(* Logix 5000 project; controller MECHATRONICS_FINAL 1769-L16ER-BB1B rev 32.11; software revision 32.00 *)

TASK MainTask (continuous, watchdog 500 ms) : MainProgram

MODULES
   Local : 1769-L16ER-BB1B (PointIO 0, rev 32.11)
      Discrete_IO : Embedded (PointIO 1, rev 32.11, Output RPI 20 ms)
END_MODULES

PROGRAM MainProgram   (* main routine MainRoutine *)
VAR
   Brakes : BOOL;
   CurrentFloor : DINT := 1;
   DoorOpen : BOOL;
   ElevatorButton : BOOL;
   EntireGarageFull : BOOL;
   FloorCapacity : INT[6] := ([0] := 8, [1] := 8, [2] := 8, [3] := 8, [4] := 8, [5] := 8);
   index : DINT;
   MotorDown : BOOL;
   MotorDownOS : BOOL;
   MotorDownTimer : TIMER := (PRE := 5000);
   MotorUp : BOOL;
   MotorUpOS : BOOL;
   MotorUpTimer : TIMER := (PRE := 5000);
   RequestArray : INT[5];
   RequestButton1 : BOOL;
   RequestButton2 : BOOL;
   RequestButton3 : BOOL;
   RequestButton4 : BOOL;
   RequestButtonBase : BOOL;
   RequestInProgress : BOOL;
   RequestOut1 : BOOL;
   RequestOut2 : BOOL;
   RequestOut3 : BOOL;
   RequestOut4 : BOOL;
   SequenceStep : DINT;
   TempVal : DINT;
   VehicleInPlace : BOOL;
   WaitTimer : TIMER := (PRE := 30000);
END_VAR

ROUTINE MainRoutine   (* ladder *)
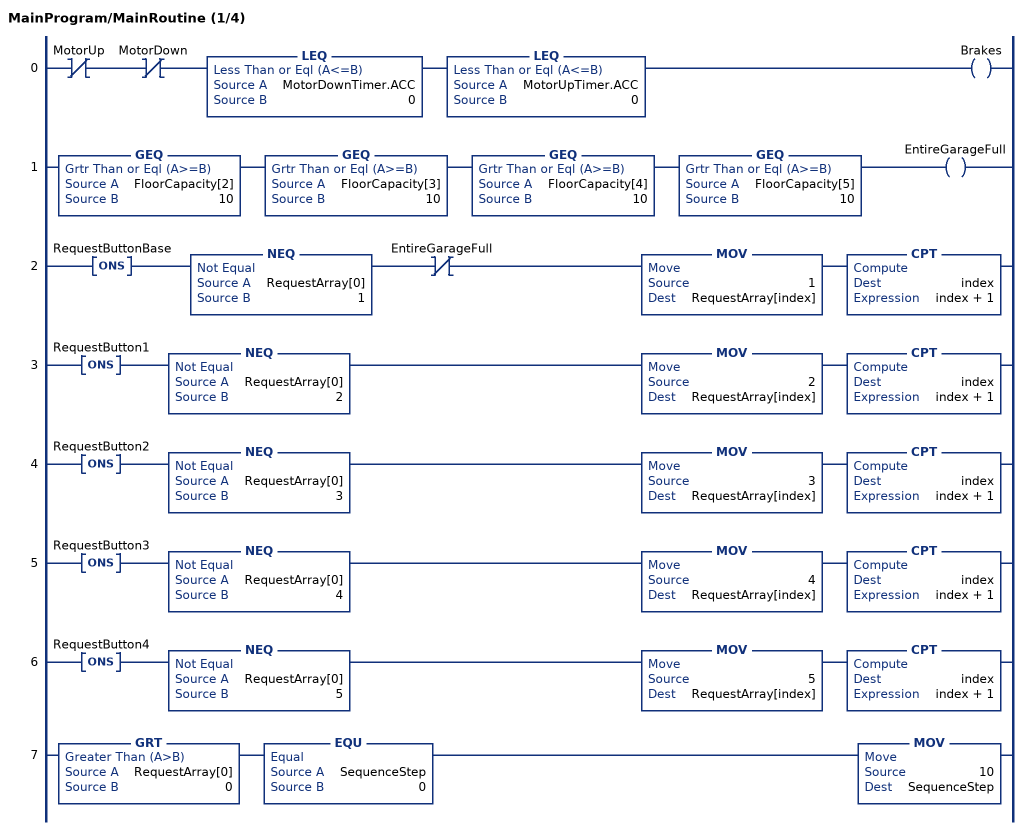
   0: XIO(MotorUp)XIO(MotorDown)LEQ(MotorDownTimer.ACC,0)LEQ(MotorUpTimer.ACC,0)OTE(Brakes);
   1: GEQ(FloorCapacity[2],10)GEQ(FloorCapacity[3],10)GEQ(FloorCapacity[4],10)GEQ(FloorCapacity[5],10)OTE(EntireGarageFull);
   2: ONS(RequestButtonBase)NEQ(RequestArray[0],1)XIO(EntireGarageFull)MOV(1,RequestArray[index])CPT(index,index + 1);
   3: ONS(RequestButton1)NEQ(RequestArray[0],2)MOV(2,RequestArray[index])CPT(index,index + 1);
   4: ONS(RequestButton2)NEQ(RequestArray[0],3)MOV(3,RequestArray[index])CPT(index,index + 1);
   5: ONS(RequestButton3)NEQ(RequestArray[0],4)MOV(4,RequestArray[index])CPT(index,index + 1);
   6: ONS(RequestButton4)NEQ(RequestArray[0],5)MOV(5,RequestArray[index])CPT(index,index + 1);
   7: GRT(RequestArray[0],0)EQU(SequenceStep,0)MOV(10,SequenceStep);
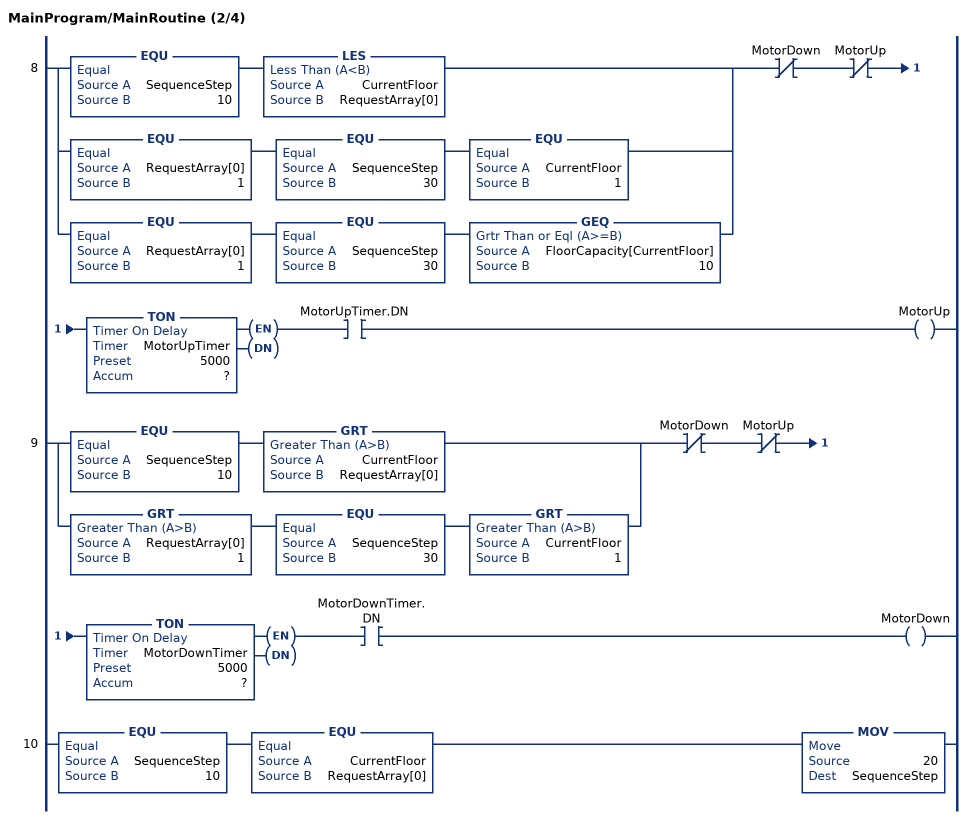
   8: [EQU(SequenceStep,10) LES(CurrentFloor,RequestArray[0]) ,[EQU(RequestArray[0],1) EQU(SequenceStep,30) EQU(CurrentFloor,1) ,EQU(RequestArray[0],1) EQU(SequenceStep,30) GEQ(FloorCapacity[CurrentFloor],10) ] ]XIO(MotorDown)XIO(MotorUp)TON(MotorUpTimer,?,?)XIC(MotorUpTimer.DN)OTE(MotorUp);
   9: [EQU(SequenceStep,10) GRT(CurrentFloor,RequestArray[0]) ,GRT(RequestArray[0],1) EQU(SequenceStep,30) GRT(CurrentFloor,1) ]XIO(MotorDown)XIO(MotorUp)TON(MotorDownTimer,?,?)XIC(MotorDownTimer.DN)OTE(MotorDown);
   10: EQU(SequenceStep,10)EQU(CurrentFloor,RequestArray[0])MOV(20,SequenceStep);
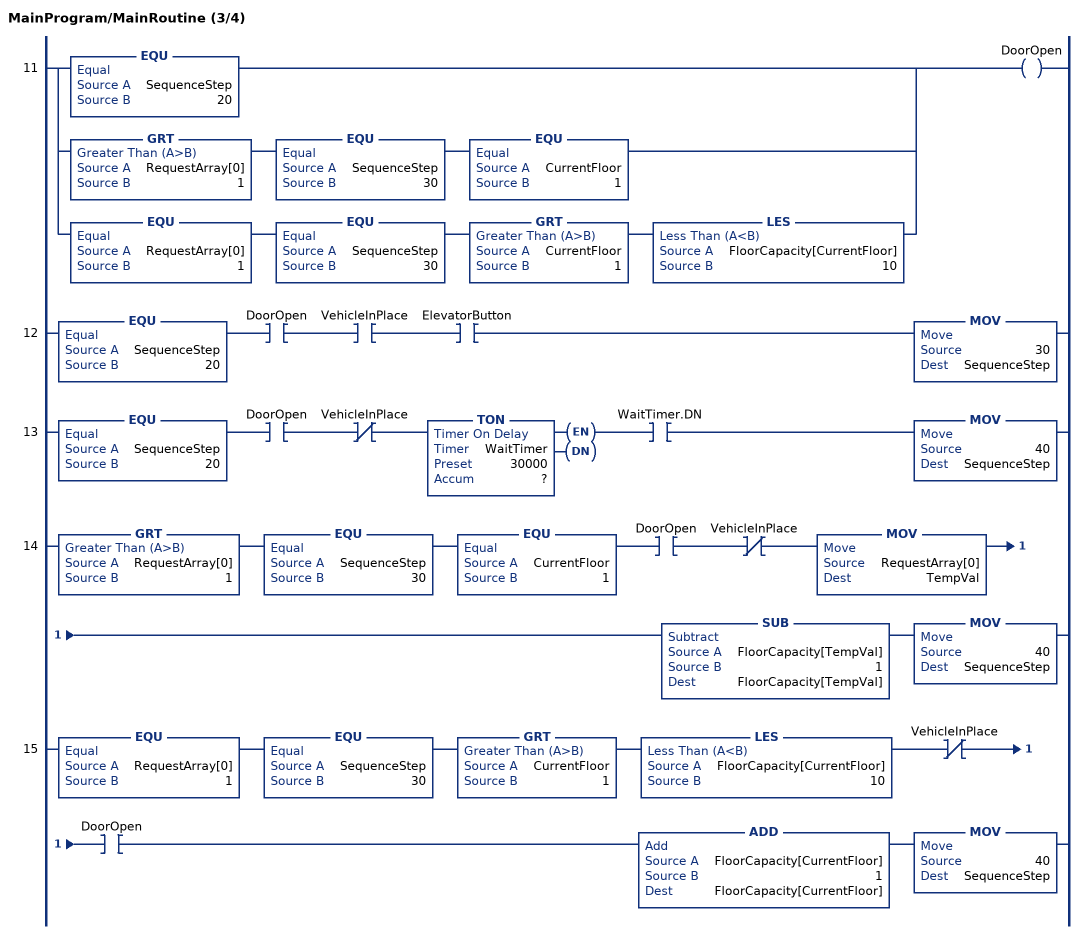
   11: [EQU(SequenceStep,20) ,[GRT(RequestArray[0],1) EQU(SequenceStep,30) EQU(CurrentFloor,1) ,EQU(RequestArray[0],1) EQU(SequenceStep,30) GRT(CurrentFloor,1) LES(FloorCapacity[CurrentFloor],10) ] ]OTE(DoorOpen);
   12: EQU(SequenceStep,20)XIC(DoorOpen)XIC(VehicleInPlace)XIC(ElevatorButton)MOV(30,SequenceStep);
   13: EQU(SequenceStep,20)XIC(DoorOpen)XIO(VehicleInPlace)TON(WaitTimer,?,?)XIC(WaitTimer.DN)MOV(40,SequenceStep);
   14: GRT(RequestArray[0],1)EQU(SequenceStep,30)EQU(CurrentFloor,1)XIC(DoorOpen)XIO(VehicleInPlace)MOV(RequestArray[0],TempVal)SUB(FloorCapacity[TempVal],1,FloorCapacity[TempVal])MOV(40,SequenceStep);
   15: EQU(RequestArray[0],1)EQU(SequenceStep,30)GRT(CurrentFloor,1)LES(FloorCapacity[CurrentFloor],10)XIO(VehicleInPlace)XIC(DoorOpen)ADD(FloorCapacity[CurrentFloor],1,FloorCapacity[CurrentFloor])MOV(40,SequenceStep);
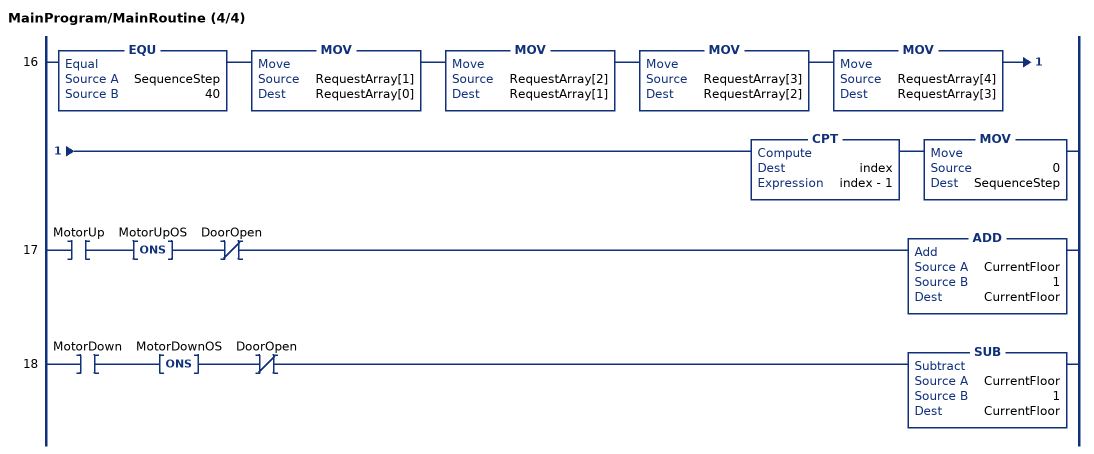
   16: EQU(SequenceStep,40)MOV(RequestArray[1],RequestArray[0])MOV(RequestArray[2],RequestArray[1])MOV(RequestArray[3],RequestArray[2])MOV(RequestArray[4],RequestArray[3])CPT(index,index - 1)MOV(0,SequenceStep);
   17: XIC(MotorUp)ONS(MotorUpOS)XIO(DoorOpen)ADD(CurrentFloor,1,CurrentFloor);
   18: XIC(MotorDown)ONS(MotorDownOS)XIO(DoorOpen)SUB(CurrentFloor,1,CurrentFloor);
END_ROUTINE
END_PROGRAM
